FUNCTION_BLOCK VentSludgeOC (* CAT Function Block Type *)
  (* Standard: 61499-2 *)
  (* Version 0.0, 6/7/2026, Schneider Electric, template *)
  PACKAGE SE.Nereda;
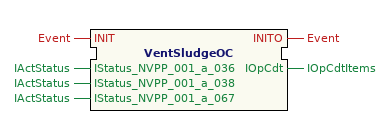
  EVENT_INPUT
    INIT;
  END_EVENT
  EVENT_OUTPUT
    INITO;
  END_EVENT
  SOCKETS
    IStatus_NVPP_001_a_036 : IActStatus;
    IStatus_NVPP_001_a_038 : IActStatus;
    IStatus_NVPP_001_a_067 : IActStatus;
  END_SOCKETS
  PLUGS
    IOpCdt : IOpCdtItems;
  END_PLUGS
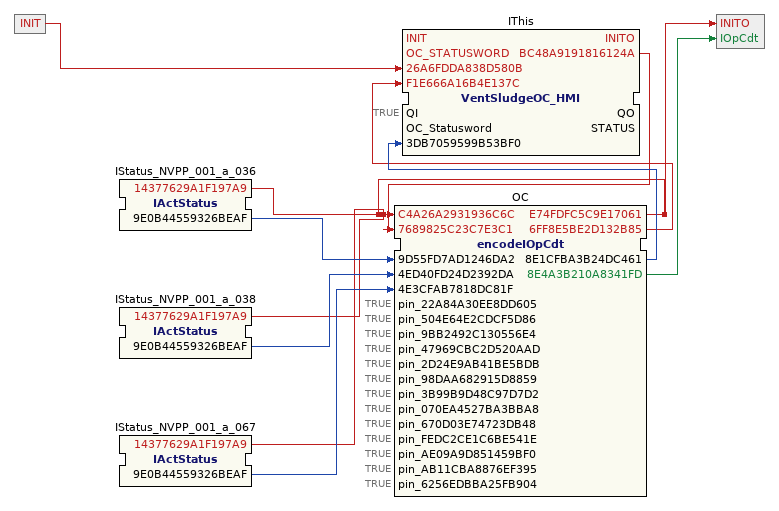
  (* 01 - FUNCTIONNAL INPUT INTERFACE *)
  (* 00 - INITIALIZATION *)
  (* 05 - LOGIC *)
  (* 06 - HMI INTERFACE *)
  (* 03 - FIELD INTERFACE *)
  (* Created by : Nouriddin OUECHEN 2026 *)
  (* Operating Condition Status *)
  (* Created by : Nouriddin OUECHEN 2026 *)
  (* 02 - FUNCTIONNAL OUTPUT INTERFACE *)
  (* Operating conditions : 1. Discharge valve NVPP 001 a-- 023 is available and valves for other reactors are closed 6. No HH-level in sludge buffer *)
  FBS
    OC : encodeIOpCdt(pin_22A84A30EE8DD605 := TRUE, pin_504E64E2CDCF5D86 := TRUE, pin_9BB2492C130556E4 := TRUE, pin_47969CBC2D520AAD := TRUE, pin_2D24E9AB41BE5BDB := TRUE, pin_98DAA682915D8859 := TRUE, pin_3B99B9D48C97D7D2 := TRUE, pin_070EA4527BA3BBA8 := TRUE, pin_670D03E74723DB48 := TRUE, pin_FEDC2CE1C6BE541E := TRUE, pin_AE09A9D851459BF0 := TRUE, pin_AB11CBA8876EF395 := TRUE, pin_6256EDBBA25FB904 := TRUE); (* You set the operating conditions. For the inputs that are not used set a constant to TRUE. *)
    IThis : VentSludgeOC_HMI(QI := TRUE);
  END_FBS
  EVENT_CONNECTIONS
    INIT TO IThis.26A6FDDA838D580B;
    IStatus_NVPP_001_a_036.14377629A1F197A9 TO OC.C4A26A2931936C6C;
    IStatus_NVPP_001_a_038.14377629A1F197A9 TO OC.C4A26A2931936C6C;
    IStatus_NVPP_001_a_067.14377629A1F197A9 TO OC.C4A26A2931936C6C;
    OC.E74FDFC5C9E17061 TO INITO;
    OC.6FF8E5BE2D132B85 TO IThis.F1E666A16B4E137C;
    IThis.BC48A9191816124A TO OC.7689825C23C7E3C1;
    OC.E74FDFC5C9E17061 TO OC.C4A26A2931936C6C;
  END_CONNECTIONS
  DATA_CONNECTIONS
    IStatus_NVPP_001_a_036.9E0B44559326BEAF TO OC.9D55FD7AD1246DA2;
    IStatus_NVPP_001_a_038.9E0B44559326BEAF TO OC.4ED40FD24D2392DA;
    IStatus_NVPP_001_a_067.9E0B44559326BEAF TO OC.4E3CFAB7818DC81F;
    OC.8E1CFBA3B24DC461 TO IThis.3DB7059599B53BF0;
  END_CONNECTIONS
  ADAPTER_CONNECTIONS
    OC.8E4A3B210A8341FD TO IOpCdt;
  END_CONNECTIONS
END_FUNCTION_BLOCK
